{attribute 'qualified_only'}
{attribute 'strict'}
TYPE E_CellState :
(
	IDLE := 0,
	WAIT_STATION := 1,
	INDEXING := 2
);
END_TYPE

(* stored: Version 1.1.0.1, ProductVersion 3.1.4024.12
   DUT E_CellState: Id {f58d99b1-5275-47d2-acf5-137e1214b895} *)
